// TIA Portal V17 export
// export: Created 2025-03-07T09:16:39.2442536Z, ExportSetting WithDefaults, DisplayName Totally Integrated Automation Portal, DisplayVersion V17 Update 8, DisplayName TIA Portal Openness, DisplayVersion V17 Update 8, DisplayName TIA Portal Version Control Interface, DisplayVersion V17, DisplayName SINAMICS Startdrive Advanced, DisplayVersion V17 SP2, DisplayName SINAMICS Startdrive G110M, G120, G120C, G120D, G120P, G115D, DisplayVersion V17 SP2, DisplayName SINAMICS Startdrive G130, G150, S120, S150, SINAMICS MV, S210, DisplayVersion V17 SP2, DisplayName STEP 7 Professional, DisplayVersion V17 Update 8, DisplayName SINUMERIK ONE STEP 7 Toolbox, DisplayVersion V17 Update 12, DisplayName SINUMERIK 840D sl STEP 7 Toolbox, DisplayVersion V17 Update 12, DisplayName STEP 7 Safety, DisplayVersion V17 Update 6, DisplayName WinCC Advanced, DisplayVersion V17 Update 8
DATA_BLOCK "DB2410_PLC_CNC_SIGNALS"   // DB2410
{ S7_Optimized_Access := 'FALSE'; DB_Accessible_From_OPC_UA := 'FALSE' }
AUTHOR : ETXETAR
VERSION : 1.0
// stored: AutoNumber false, DBAccessibleFromOPCUA false, DBAccessibleFromWebserver true, IsOnlyStoredInLoadMemory false, IsWriteProtectedInAS false
   VAR RETAIN
      PLC_NC_SIGNALS_1_32 : Struct   // NCK INPUTS EXTENSION BIT 41-72 / PLC NC SIGNALS BIT 1-32
         PLC_NC_SIGNAL_1 : Bool;   // NCK INPUTS EXTENSION 41 / PLC NC SIGNAL 1
         PLC_NC_SIGNAL_2 : Bool;   // NCK INPUTS EXTENSION 42 / PLC NC SIGNAL 2
         PLC_NC_SIGNAL_3 : Bool;   // NCK INPUTS EXTENSION 43 / PLC NC SIGNAL 3
         PLC_NC_SIGNAL_4 : Bool;   // NCK INPUTS EXTENSION 44 / PLC NC SIGNAL 4
         PLC_NC_SIGNAL_5 : Bool;   // NCK INPUTS EXTENSION 45 / PLC NC SIGNAL 5
         PLC_NC_SIGNAL_6 : Bool;   // NCK INPUTS EXTENSION 46 / PLC NC SIGNAL 6
         PLC_NC_SIGNAL_7 : Bool;   // NCK INPUTS EXTENSION 47 / PLC NC SIGNAL 7
         PLC_NC_SIGNAL_8 : Bool;   // NCK INPUTS EXTENSION 48 / PLC NC SIGNAL 8
         PLC_NC_SIGNAL_9 : Bool;   // NCK INPUTS EXTENSION 49 / PLC NC SIGNAL 9
         PLC_NC_SIGNAL_10 : Bool;   // NCK INPUTS EXTENSION 50 / PLC NC SIGNAL 10
         PLC_NC_SIGNAL_11 : Bool;   // NCK INPUTS EXTENSION 51 / PLC NC SIGNAL 11
         PLC_NC_SIGNAL_12 : Bool;   // NCK INPUTS EXTENSION 52 / PLC NC SIGNAL 12
         PLC_NC_SIGNAL_13 : Bool;   // NCK INPUTS EXTENSION 53 / PLC NC SIGNAL 13
         PLC_NC_SIGNAL_14 : Bool;   // NCK INPUTS EXTENSION 54 / PLC NC SIGNAL 14
         PLC_NC_SIGNAL_15 : Bool;   // NCK INPUTS EXTENSION 55 / PLC NC SIGNAL 15
         PLC_NC_SIGNAL_16 : Bool;   // NCK INPUTS EXTENSION 56 / PLC NC SIGNAL 16
         PLC_NC_SIGNAL_17 : Bool;   // NCK INPUTS EXTENSION 57 / PLC NC SIGNAL 17
         PLC_NC_SIGNAL_18 : Bool;   // NCK INPUTS EXTENSION 58 / PLC NC SIGNAL 18
         PLC_NC_SIGNAL_19 : Bool;   // NCK INPUTS EXTENSION 59 / PLC NC SIGNAL 19
         PLC_NC_SIGNAL_20 : Bool;   // NCK INPUTS EXTENSION 60 / PLC NC SIGNAL 20
         PLC_NC_SIGNAL_21 : Bool;   // NCK INPUTS EXTENSION 61 / PLC NC SIGNAL 21
         PLC_NC_SIGNAL_22 : Bool;   // NCK INPUTS EXTENSION 62 / PLC NC SIGNAL 22
         PLC_NC_SIGNAL_23 : Bool;   // NCK INPUTS EXTENSION 63 / PLC NC SIGNAL 23
         PLC_NC_SIGNAL_24 : Bool;   // NCK INPUTS EXTENSION 64 / PLC NC SIGNAL 24
         PLC_NC_SIGNAL_25 : Bool;   // NCK INPUTS EXTENSION 65 / PLC NC SIGNAL 25
         PLC_NC_SIGNAL_26 : Bool;   // NCK INPUTS EXTENSION 66 / PLC NC SIGNAL 26
         PLC_NC_SIGNAL_27 : Bool;   // NCK INPUTS EXTENSION 67 / PLC NC SIGNAL 27
         PLC_NC_SIGNAL_28 : Bool;   // NCK INPUTS EXTENSION 68 / PLC NC SIGNAL 28
         PLC_NC_SIGNAL_29 : Bool;   // NCK INPUTS EXTENSION 69 / PLC NC SIGNAL 29
         PLC_NC_SIGNAL_30 : Bool;   // NCK INPUTS EXTENSION 70 / PLC NC SIGNAL 30
         PLC_NC_SIGNAL_31 : Bool;   // NCK INPUTS EXTENSION 71 / PLC NC SIGNAL 31
         PLC_NC_SIGNAL_32 : Bool;   // NCK INPUTS EXTENSION 72 / PLC NC SIGNAL 32
      END_STRUCT;
      PLC_NC_SIGNALS_33_64 : Struct   // NCK INPUTS EXTENSION BIT 73-104 / PLC NC SIGNALS BIT 33-64
         PLC_NC_SIGNAL_33 : Bool;   // NCK INPUTS EXTENSION 73 / PLC NC SIGNAL 33
         PLC_NC_SIGNAL_34 : Bool;   // NCK INPUTS EXTENSION 74 / PLC NC SIGNAL 34
         PLC_NC_SIGNAL_35 : Bool;   // NCK INPUTS EXTENSION 75 / PLC NC SIGNAL 35
         PLC_NC_SIGNAL_36 : Bool;   // NCK INPUTS EXTENSION 76 / PLC NC SIGNAL 36
         PLC_NC_SIGNAL_37 : Bool;   // NCK INPUTS EXTENSION 77 / PLC NC SIGNAL 37
         PLC_NC_SIGNAL_38 : Bool;   // NCK INPUTS EXTENSION 78 / PLC NC SIGNAL 38
         PLC_NC_SIGNAL_39 : Bool;   // NCK INPUTS EXTENSION 79 / PLC NC SIGNAL 39
         PLC_NC_SIGNAL_40 : Bool;   // NCK INPUTS EXTENSION 80 / PLC NC SIGNAL 40
         PLC_NC_SIGNAL_41 : Bool;   // NCK INPUTS EXTENSION 81 / PLC NC SIGNAL 41
         PLC_NC_SIGNAL_42 : Bool;   // NCK INPUTS EXTENSION 82 / PLC NC SIGNAL 42
         PLC_NC_SIGNAL_43 : Bool;   // NCK INPUTS EXTENSION 83 / PLC NC SIGNAL 43
         PLC_NC_SIGNAL_44 : Bool;   // NCK INPUTS EXTENSION 84 / PLC NC SIGNAL 44
         PLC_NC_SIGNAL_45 : Bool;   // NCK INPUTS EXTENSION 85 / PLC NC SIGNAL 45
         PLC_NC_SIGNAL_46 : Bool;   // NCK INPUTS EXTENSION 86 / PLC NC SIGNAL 46
         PLC_NC_SIGNAL_47 : Bool;   // NCK INPUTS EXTENSION 87 / PLC NC SIGNAL 47
         PLC_NC_SIGNAL_48 : Bool;   // NCK INPUTS EXTENSION 88 / PLC NC SIGNAL 48
         PLC_NC_SIGNAL_49 : Bool;   // NCK INPUTS EXTENSION 89 / PLC NC SIGNAL 49
         PLC_NC_SIGNAL_50 : Bool;   // NCK INPUTS EXTENSION 90 / PLC NC SIGNAL 50
         PLC_NC_SIGNAL_51 : Bool;   // NCK INPUTS EXTENSION 91 / PLC NC SIGNAL 51
         PLC_NC_SIGNAL_52 : Bool;   // NCK INPUTS EXTENSION 92 / PLC NC SIGNAL 52
         PLC_NC_SIGNAL_53 : Bool;   // NCK INPUTS EXTENSION 93 / PLC NC SIGNAL 53
         PLC_NC_SIGNAL_54 : Bool;   // NCK INPUTS EXTENSION 94 / PLC NC SIGNAL 54
         PLC_NC_SIGNAL_55 : Bool;   // NCK INPUTS EXTENSION 95 / PLC NC SIGNAL 55
         PLC_NC_SIGNAL_56 : Bool;   // NCK INPUTS EXTENSION 96 / PLC NC SIGNAL 56
         PLC_NC_SIGNAL_57 : Bool;   // NCK INPUTS EXTENSION 97 / PLC NC SIGNAL 57
         PLC_NC_SIGNAL_58 : Bool;   // NCK INPUTS EXTENSION 98 / PLC NC SIGNAL 58
         PLC_NC_SIGNAL_59 : Bool;   // NCK INPUTS EXTENSION 99 / PLC NC SIGNAL 59
         PLC_NC_SIGNAL_60 : Bool;   // NCK INPUTS EXTENSION 100 / PLC NC SIGNAL 60
         PLC_NC_SIGNAL_61 : Bool;   // NCK INPUTS EXTENSION 101 / PLC NC SIGNAL 61
         PLC_NC_SIGNAL_62 : Bool;   // NCK INPUTS EXTENSION 102 / PLC NC SIGNAL 62
         PLC_NC_SIGNAL_63 : Bool;   // NCK INPUTS EXTENSION 103 / PLC NC SIGNAL 63
         PLC_NC_SIGNAL_64 : Bool;   // NCK INPUTS EXTENSION 104 / PLC NC SIGNAL 64
      END_STRUCT;
      PLC_NC_SIGNALS_65_96 : Struct   // NCK INPUTS EXTENSION BIT 73-104 / PLC NC SIGNALS BIT 65-96
         PLC_NC_SIGNAL_65 : Bool;   // NCK INPUTS EXTENSION 73 / PLC NC SIGNAL 65
         PLC_NC_SIGNAL_66 : Bool;   // NCK INPUTS EXTENSION 74 / PLC NC SIGNAL 66
         PLC_NC_SIGNAL_67 : Bool;   // NCK INPUTS EXTENSION 75 / PLC NC SIGNAL 67
         PLC_NC_SIGNAL_68 : Bool;   // NCK INPUTS EXTENSION 76 / PLC NC SIGNAL 68
         PLC_NC_SIGNAL_69 : Bool;   // NCK INPUTS EXTENSION 77 / PLC NC SIGNAL 69
         PLC_NC_SIGNAL_70 : Bool;   // NCK INPUTS EXTENSION 78 / PLC NC SIGNAL 70
         PLC_NC_SIGNAL_71 : Bool;   // NCK INPUTS EXTENSION 79 / PLC NC SIGNAL 71
         PLC_NC_SIGNAL_72 : Bool;   // NCK INPUTS EXTENSION 80 / PLC NC SIGNAL 72
         PLC_NC_SIGNAL_73 : Bool;   // NCK INPUTS EXTENSION 81 / PLC NC SIGNAL 73
         PLC_NC_SIGNAL_74 : Bool;   // NCK INPUTS EXTENSION 82 / PLC NC SIGNAL 74
         PLC_NC_SIGNAL_75 : Bool;   // NCK INPUTS EXTENSION 83 / PLC NC SIGNAL 75
         PLC_NC_SIGNAL_76 : Bool;   // NCK INPUTS EXTENSION 84 / PLC NC SIGNAL 76
         PLC_NC_SIGNAL_77 : Bool;   // NCK INPUTS EXTENSION 85 / PLC NC SIGNAL 77
         PLC_NC_SIGNAL_78 : Bool;   // NCK INPUTS EXTENSION 86 / PLC NC SIGNAL 78
         PLC_NC_SIGNAL_79 : Bool;   // NCK INPUTS EXTENSION 87 / PLC NC SIGNAL 79
         PLC_NC_SIGNAL_80 : Bool;   // NCK INPUTS EXTENSION 88 / PLC NC SIGNAL 80
         PLC_NC_SIGNAL_81 : Bool;   // NCK INPUTS EXTENSION 89 / PLC NC SIGNAL 81
         PLC_NC_SIGNAL_82 : Bool;   // NCK INPUTS EXTENSION 90 / PLC NC SIGNAL 82
         PLC_NC_SIGNAL_83 : Bool;   // NCK INPUTS EXTENSION 91 / PLC NC SIGNAL 83
         PLC_NC_SIGNAL_84 : Bool;   // NCK INPUTS EXTENSION 92 / PLC NC SIGNAL 84
         PLC_NC_SIGNAL_85 : Bool;   // NCK INPUTS EXTENSION 93 / PLC NC SIGNAL 85
         PLC_NC_SIGNAL_86 : Bool;   // NCK INPUTS EXTENSION 94 / PLC NC SIGNAL 86
         PLC_NC_SIGNAL_87 : Bool;   // NCK INPUTS EXTENSION 95 / PLC NC SIGNAL 87
         PLC_NC_SIGNAL_88 : Bool;   // NCK INPUTS EXTENSION 96 / PLC NC SIGNAL 88
         PLC_NC_SIGNAL_89 : Bool;   // NCK INPUTS EXTENSION 97 / PLC NC SIGNAL 89
         PLC_NC_SIGNAL_90 : Bool;   // NCK INPUTS EXTENSION 98 / PLC NC SIGNAL 90
         PLC_NC_SIGNAL_91 : Bool;   // NCK INPUTS EXTENSION 99 / PLC NC SIGNAL 91
         PLC_NC_SIGNAL_92 : Bool;   // NCK INPUTS EXTENSION 100 / PLC NC SIGNAL 92
         PLC_NC_SIGNAL_93 : Bool;   // NCK INPUTS EXTENSION 101 / PLC NC SIGNAL 93
         PLC_NC_SIGNAL_94 : Bool;   // NCK INPUTS EXTENSION 102 / PLC NC SIGNAL 94
         PLC_NC_SIGNAL_95 : Bool;   // NCK INPUTS EXTENSION 103 / PLC NC SIGNAL 95
         PLC_NC_SIGNAL_96 : Bool;   // NCK INPUTS EXTENSION 104 / PLC NC SIGNAL 96
      END_STRUCT;
      PLC_NC_SIGNALS_97_128 : Struct   // NCK INPUTS EXTENSION BIT 73-104 / PLC NC SIGNALS BIT 97-128
         PLC_NC_SIGNAL_97 : Bool;   // NCK INPUTS EXTENSION 73 / PLC NC SIGNAL 97
         PLC_NC_SIGNAL_98 : Bool;   // NCK INPUTS EXTENSION 74 / PLC NC SIGNAL 98
         PLC_NC_SIGNAL_99 : Bool;   // NCK INPUTS EXTENSION 75 / PLC NC SIGNAL 99
         PLC_NC_SIGNAL_100 : Bool;   // NCK INPUTS EXTENSION 76 / PLC NC SIGNAL 100
         PLC_NC_SIGNAL_101 : Bool;   // NCK INPUTS EXTENSION 77 / PLC NC SIGNAL 101
         PLC_NC_SIGNAL_102 : Bool;   // NCK INPUTS EXTENSION 78 / PLC NC SIGNAL 102
         PLC_NC_SIGNAL_103 : Bool;   // NCK INPUTS EXTENSION 79 / PLC NC SIGNAL 103
         PLC_NC_SIGNAL_104 : Bool;   // NCK INPUTS EXTENSION 80 / PLC NC SIGNAL 104
         PLC_NC_SIGNAL_105 : Bool;   // NCK INPUTS EXTENSION 81 / PLC NC SIGNAL 105
         PLC_NC_SIGNAL_106 : Bool;   // NCK INPUTS EXTENSION 82 / PLC NC SIGNAL 106
         PLC_NC_SIGNAL_107 : Bool;   // NCK INPUTS EXTENSION 83 / PLC NC SIGNAL 107
         PLC_NC_SIGNAL_108 : Bool;   // NCK INPUTS EXTENSION 84 / PLC NC SIGNAL 108
         PLC_NC_SIGNAL_109 : Bool;   // NCK INPUTS EXTENSION 85 / PLC NC SIGNAL 109
         PLC_NC_SIGNAL_110 : Bool;   // NCK INPUTS EXTENSION 86 / PLC NC SIGNAL 110
         PLC_NC_SIGNAL_111 : Bool;   // NCK INPUTS EXTENSION 87 / PLC NC SIGNAL 111
         PLC_NC_SIGNAL_112 : Bool;   // NCK INPUTS EXTENSION 88 / PLC NC SIGNAL 112
         PLC_NC_SIGNAL_113 : Bool;   // NCK INPUTS EXTENSION 89 / PLC NC SIGNAL 113
         PLC_NC_SIGNAL_114 : Bool;   // NCK INPUTS EXTENSION 90 / PLC NC SIGNAL 114
         PLC_NC_SIGNAL_115 : Bool;   // NCK INPUTS EXTENSION 91 / PLC NC SIGNAL 115
         PLC_NC_SIGNAL_116 : Bool;   // NCK INPUTS EXTENSION 92 / PLC NC SIGNAL 116
         PLC_NC_SIGNAL_117 : Bool;   // NCK INPUTS EXTENSION 93 / PLC NC SIGNAL 117
         PLC_NC_SIGNAL_118 : Bool;   // NCK INPUTS EXTENSION 94 / PLC NC SIGNAL 118
         PLC_NC_SIGNAL_119 : Bool;   // NCK INPUTS EXTENSION 95 / PLC NC SIGNAL 119
         PLC_NC_SIGNAL_120 : Bool;   // NCK INPUTS EXTENSION 96 / PLC NC SIGNAL 120
         PLC_NC_SIGNAL_121 : Bool;   // NCK INPUTS EXTENSION 97 / PLC NC SIGNAL 121
         PLC_NC_SIGNAL_122 : Bool;   // NCK INPUTS EXTENSION 98 / PLC NC SIGNAL 122
         PLC_NC_SIGNAL_123 : Bool;   // NCK INPUTS EXTENSION 99 / PLC NC SIGNAL 123
         PLC_NC_SIGNAL_124 : Bool;   // NCK INPUTS EXTENSION 100 / PLC NC SIGNAL 124
         PLC_NC_SIGNAL_125 : Bool;   // NCK INPUTS EXTENSION 101 / PLC NC SIGNAL 125
         PLC_NC_SIGNAL_126 : Bool;   // NCK INPUTS EXTENSION 102 / PLC NC SIGNAL 126
         PLC_NC_SIGNAL_127 : Bool;   // NCK INPUTS EXTENSION 103 / PLC NC SIGNAL 127
         PLC_NC_SIGNAL_128 : Bool;   // NCK INPUTS EXTENSION 104 / PLC NC SIGNAL 128
      END_STRUCT;
      PLC_NC_SIGNALS_129_160 : Struct   // NCK INPUTS EXTENSION BIT 73-104 / PLC NC SIGNALS BIT 129-160
         PLC_NC_SIGNAL_129 : Bool;   // NCK INPUTS EXTENSION 73 / PLC NC SIGNAL 129
         PLC_NC_SIGNAL_130 : Bool;   // NCK INPUTS EXTENSION 74 / PLC NC SIGNAL 130
         PLC_NC_SIGNAL_131 : Bool;   // NCK INPUTS EXTENSION 75 / PLC NC SIGNAL 131
         PLC_NC_SIGNAL_132 : Bool;   // NCK INPUTS EXTENSION 76 / PLC NC SIGNAL 132
         PLC_NC_SIGNAL_133 : Bool;   // NCK INPUTS EXTENSION 77 / PLC NC SIGNAL 133
         PLC_NC_SIGNAL_134 : Bool;   // NCK INPUTS EXTENSION 78 / PLC NC SIGNAL 134
         PLC_NC_SIGNAL_135 : Bool;   // NCK INPUTS EXTENSION 79 / PLC NC SIGNAL 135
         PLC_NC_SIGNAL_136 : Bool;   // NCK INPUTS EXTENSION 80 / PLC NC SIGNAL 136
         PLC_NC_SIGNAL_137 : Bool;   // NCK INPUTS EXTENSION 81 / PLC NC SIGNAL 137
         PLC_NC_SIGNAL_138 : Bool;   // NCK INPUTS EXTENSION 82 / PLC NC SIGNAL 138
         PLC_NC_SIGNAL_139 : Bool;   // NCK INPUTS EXTENSION 83 / PLC NC SIGNAL 139
         PLC_NC_SIGNAL_140 : Bool;   // NCK INPUTS EXTENSION 84 / PLC NC SIGNAL 140
         PLC_NC_SIGNAL_141 : Bool;   // NCK INPUTS EXTENSION 85 / PLC NC SIGNAL 141
         PLC_NC_SIGNAL_142 : Bool;   // NCK INPUTS EXTENSION 86 / PLC NC SIGNAL 142
         PLC_NC_SIGNAL_143 : Bool;   // NCK INPUTS EXTENSION 87 / PLC NC SIGNAL 143
         PLC_NC_SIGNAL_144 : Bool;   // NCK INPUTS EXTENSION 88 / PLC NC SIGNAL 144
         PLC_NC_SIGNAL_145 : Bool;   // NCK INPUTS EXTENSION 89 / PLC NC SIGNAL 145
         PLC_NC_SIGNAL_146 : Bool;   // NCK INPUTS EXTENSION 90 / PLC NC SIGNAL 146
         PLC_NC_SIGNAL_147 : Bool;   // NCK INPUTS EXTENSION 91 / PLC NC SIGNAL 147
         PLC_NC_SIGNAL_148 : Bool;   // NCK INPUTS EXTENSION 92 / PLC NC SIGNAL 148
         PLC_NC_SIGNAL_149 : Bool;   // NCK INPUTS EXTENSION 93 / PLC NC SIGNAL 149
         PLC_NC_SIGNAL_150 : Bool;   // NCK INPUTS EXTENSION 94 / PLC NC SIGNAL 150
         PLC_NC_SIGNAL_151 : Bool;   // NCK INPUTS EXTENSION 95 / PLC NC SIGNAL 151
         PLC_NC_SIGNAL_152 : Bool;   // NCK INPUTS EXTENSION 96 / PLC NC SIGNAL 152
         PLC_NC_SIGNAL_153 : Bool;   // NCK INPUTS EXTENSION 97 / PLC NC SIGNAL 153
         PLC_NC_SIGNAL_154 : Bool;   // NCK INPUTS EXTENSION 98 / PLC NC SIGNAL 154
         PLC_NC_SIGNAL_155 : Bool;   // NCK INPUTS EXTENSION 99 / PLC NC SIGNAL 155
         PLC_NC_SIGNAL_156 : Bool;   // NCK INPUTS EXTENSION 100 / PLC NC SIGNAL 156
         PLC_NC_SIGNAL_157 : Bool;   // NCK INPUTS EXTENSION 101 / PLC NC SIGNAL 157
         PLC_NC_SIGNAL_158 : Bool;   // NCK INPUTS EXTENSION 102 / PLC NC SIGNAL 158
         PLC_NC_SIGNAL_159 : Bool;   // NCK INPUTS EXTENSION 103 / PLC NC SIGNAL 159
         PLC_NC_SIGNAL_160 : Bool;   // NCK INPUTS EXTENSION 104 / PLC NC SIGNAL 160
      END_STRUCT;
      PLC_NC_SIGNALS_161_192 : Struct   // NCK INPUTS EXTENSION BIT 73-104 / PLC NC SIGNALS BIT 161-192
         PLC_NC_SIGNAL_161 : Bool;   // NCK INPUTS EXTENSION 73 / PLC NC SIGNAL 161
         PLC_NC_SIGNAL_162 : Bool;   // NCK INPUTS EXTENSION 74 / PLC NC SIGNAL 162
         PLC_NC_SIGNAL_163 : Bool;   // NCK INPUTS EXTENSION 75 / PLC NC SIGNAL 163
         PLC_NC_SIGNAL_164 : Bool;   // NCK INPUTS EXTENSION 76 / PLC NC SIGNAL 164
         PLC_NC_SIGNAL_165 : Bool;   // NCK INPUTS EXTENSION 77 / PLC NC SIGNAL 165
         PLC_NC_SIGNAL_166 : Bool;   // NCK INPUTS EXTENSION 78 / PLC NC SIGNAL 166
         PLC_NC_SIGNAL_167 : Bool;   // NCK INPUTS EXTENSION 79 / PLC NC SIGNAL 167
         PLC_NC_SIGNAL_168 : Bool;   // NCK INPUTS EXTENSION 80 / PLC NC SIGNAL 168
         PLC_NC_SIGNAL_169 : Bool;   // NCK INPUTS EXTENSION 81 / PLC NC SIGNAL 169
         PLC_NC_SIGNAL_170 : Bool;   // NCK INPUTS EXTENSION 82 / PLC NC SIGNAL 170
         PLC_NC_SIGNAL_171 : Bool;   // NCK INPUTS EXTENSION 83 / PLC NC SIGNAL 171
         PLC_NC_SIGNAL_172 : Bool;   // NCK INPUTS EXTENSION 84 / PLC NC SIGNAL 172
         PLC_NC_SIGNAL_173 : Bool;   // NCK INPUTS EXTENSION 85 / PLC NC SIGNAL 173
         PLC_NC_SIGNAL_174 : Bool;   // NCK INPUTS EXTENSION 86 / PLC NC SIGNAL 174
         PLC_NC_SIGNAL_175 : Bool;   // NCK INPUTS EXTENSION 87 / PLC NC SIGNAL 175
         PLC_NC_SIGNAL_176 : Bool;   // NCK INPUTS EXTENSION 88 / PLC NC SIGNAL 176
         PLC_NC_SIGNAL_177 : Bool;   // NCK INPUTS EXTENSION 89 / PLC NC SIGNAL 177
         PLC_NC_SIGNAL_178 : Bool;   // NCK INPUTS EXTENSION 90 / PLC NC SIGNAL 178
         PLC_NC_SIGNAL_179 : Bool;   // NCK INPUTS EXTENSION 91 / PLC NC SIGNAL 179
         PLC_NC_SIGNAL_180 : Bool;   // NCK INPUTS EXTENSION 92 / PLC NC SIGNAL 180
         PLC_NC_SIGNAL_181 : Bool;   // NCK INPUTS EXTENSION 93 / PLC NC SIGNAL 181
         PLC_NC_SIGNAL_182 : Bool;   // NCK INPUTS EXTENSION 94 / PLC NC SIGNAL 182
         PLC_NC_SIGNAL_183 : Bool;   // NCK INPUTS EXTENSION 95 / PLC NC SIGNAL 183
         PLC_NC_SIGNAL_184 : Bool;   // NCK INPUTS EXTENSION 96 / PLC NC SIGNAL 184
         PLC_NC_SIGNAL_185 : Bool;   // NCK INPUTS EXTENSION 97 / PLC NC SIGNAL 185
         PLC_NC_SIGNAL_186 : Bool;   // NCK INPUTS EXTENSION 98 / PLC NC SIGNAL 186
         PLC_NC_SIGNAL_187 : Bool;   // NCK INPUTS EXTENSION 99 / PLC NC SIGNAL 187
         PLC_NC_SIGNAL_188 : Bool;   // NCK INPUTS EXTENSION 100 / PLC NC SIGNAL 188
         PLC_NC_SIGNAL_189 : Bool;   // NCK INPUTS EXTENSION 101 / PLC NC SIGNAL 189
         PLC_NC_SIGNAL_190 : Bool;   // NCK INPUTS EXTENSION 102 / PLC NC SIGNAL 190
         PLC_NC_SIGNAL_191 : Bool;   // NCK INPUTS EXTENSION 103 / PLC NC SIGNAL 191
         PLC_NC_SIGNAL_192 : Bool;   // NCK INPUTS EXTENSION 104 / PLC NC SIGNAL 192
      END_STRUCT;
      PLC_NC_SIGNALS_193_224 : Struct   // NCK INPUTS EXTENSION BIT 73-104 / PLC NC SIGNALS BIT 193-224
         PLC_NC_SIGNAL_193 : Bool;   // NCK INPUTS EXTENSION 73 / PLC NC SIGNAL 193
         PLC_NC_SIGNAL_194 : Bool;   // NCK INPUTS EXTENSION 74 / PLC NC SIGNAL 194
         PLC_NC_SIGNAL_195 : Bool;   // NCK INPUTS EXTENSION 75 / PLC NC SIGNAL 195
         PLC_NC_SIGNAL_196 : Bool;   // NCK INPUTS EXTENSION 76 / PLC NC SIGNAL 196
         PLC_NC_SIGNAL_197 : Bool;   // NCK INPUTS EXTENSION 77 / PLC NC SIGNAL 197
         PLC_NC_SIGNAL_198 : Bool;   // NCK INPUTS EXTENSION 78 / PLC NC SIGNAL 198
         PLC_NC_SIGNAL_199 : Bool;   // NCK INPUTS EXTENSION 79 / PLC NC SIGNAL 199
         PLC_NC_SIGNAL_200 : Bool;   // NCK INPUTS EXTENSION 80 / PLC NC SIGNAL 200
         PLC_NC_SIGNAL_201 : Bool;   // NCK INPUTS EXTENSION 81 / PLC NC SIGNAL 201
         PLC_NC_SIGNAL_202 : Bool;   // NCK INPUTS EXTENSION 82 / PLC NC SIGNAL 202
         PLC_NC_SIGNAL_203 : Bool;   // NCK INPUTS EXTENSION 83 / PLC NC SIGNAL 203
         PLC_NC_SIGNAL_204 : Bool;   // NCK INPUTS EXTENSION 84 / PLC NC SIGNAL 204
         PLC_NC_SIGNAL_205 : Bool;   // NCK INPUTS EXTENSION 85 / PLC NC SIGNAL 205
         PLC_NC_SIGNAL_206 : Bool;   // NCK INPUTS EXTENSION 86 / PLC NC SIGNAL 206
         PLC_NC_SIGNAL_207 : Bool;   // NCK INPUTS EXTENSION 87 / PLC NC SIGNAL 207
         PLC_NC_SIGNAL_208 : Bool;   // NCK INPUTS EXTENSION 88 / PLC NC SIGNAL 208
         PLC_NC_SIGNAL_209 : Bool;   // NCK INPUTS EXTENSION 89 / PLC NC SIGNAL 209
         PLC_NC_SIGNAL_210 : Bool;   // NCK INPUTS EXTENSION 90 / PLC NC SIGNAL 210
         PLC_NC_SIGNAL_211 : Bool;   // NCK INPUTS EXTENSION 91 / PLC NC SIGNAL 211
         PLC_NC_SIGNAL_212 : Bool;   // NCK INPUTS EXTENSION 92 / PLC NC SIGNAL 212
         PLC_NC_SIGNAL_213 : Bool;   // NCK INPUTS EXTENSION 93 / PLC NC SIGNAL 213
         PLC_NC_SIGNAL_214 : Bool;   // NCK INPUTS EXTENSION 94 / PLC NC SIGNAL 214
         PLC_NC_SIGNAL_215 : Bool;   // NCK INPUTS EXTENSION 95 / PLC NC SIGNAL 215
         PLC_NC_SIGNAL_216 : Bool;   // NCK INPUTS EXTENSION 96 / PLC NC SIGNAL 216
         PLC_NC_SIGNAL_217 : Bool;   // NCK INPUTS EXTENSION 97 / PLC NC SIGNAL 217
         PLC_NC_SIGNAL_218 : Bool;   // NCK INPUTS EXTENSION 98 / PLC NC SIGNAL 218
         PLC_NC_SIGNAL_219 : Bool;   // NCK INPUTS EXTENSION 99 / PLC NC SIGNAL 219
         PLC_NC_SIGNAL_220 : Bool;   // NCK INPUTS EXTENSION 100 / PLC NC SIGNAL 220
         PLC_NC_SIGNAL_221 : Bool;   // NCK INPUTS EXTENSION 101 / PLC NC SIGNAL 221
         PLC_NC_SIGNAL_222 : Bool;   // NCK INPUTS EXTENSION 102 / PLC NC SIGNAL 222
         PLC_NC_SIGNAL_223 : Bool;   // NCK INPUTS EXTENSION 103 / PLC NC SIGNAL 223
         PLC_NC_SIGNAL_224 : Bool;   // NCK INPUTS EXTENSION 104 / PLC NC SIGNAL 224
      END_STRUCT;
      PLC_NC_SIGNALS_225_256 : Struct   // NCK INPUTS EXTENSION BIT 73-104 / PLC NC SIGNALS BIT 225-256
         PLC_NC_SIGNAL_225 : Bool;   // NCK INPUTS EXTENSION 73 / PLC NC SIGNAL 225
         PLC_NC_SIGNAL_226 : Bool;   // NCK INPUTS EXTENSION 74 / PLC NC SIGNAL 226
         PLC_NC_SIGNAL_227 : Bool;   // NCK INPUTS EXTENSION 75 / PLC NC SIGNAL 227
         PLC_NC_SIGNAL_228 : Bool;   // NCK INPUTS EXTENSION 76 / PLC NC SIGNAL 228
         PLC_NC_SIGNAL_229 : Bool;   // NCK INPUTS EXTENSION 77 / PLC NC SIGNAL 229
         PLC_NC_SIGNAL_230 : Bool;   // NCK INPUTS EXTENSION 78 / PLC NC SIGNAL 230
         PLC_NC_SIGNAL_231 : Bool;   // NCK INPUTS EXTENSION 79 / PLC NC SIGNAL 231
         PLC_NC_SIGNAL_232 : Bool;   // NCK INPUTS EXTENSION 80 / PLC NC SIGNAL 232
         PLC_NC_SIGNAL_233 : Bool;   // NCK INPUTS EXTENSION 81 / PLC NC SIGNAL 233
         PLC_NC_SIGNAL_234 : Bool;   // NCK INPUTS EXTENSION 82 / PLC NC SIGNAL 234
         PLC_NC_SIGNAL_235 : Bool;   // NCK INPUTS EXTENSION 83 / PLC NC SIGNAL 235
         PLC_NC_SIGNAL_236 : Bool;   // NCK INPUTS EXTENSION 84 / PLC NC SIGNAL 236
         PLC_NC_SIGNAL_237 : Bool;   // NCK INPUTS EXTENSION 85 / PLC NC SIGNAL 237
         PLC_NC_SIGNAL_238 : Bool;   // NCK INPUTS EXTENSION 86 / PLC NC SIGNAL 238
         PLC_NC_SIGNAL_239 : Bool;   // NCK INPUTS EXTENSION 87 / PLC NC SIGNAL 239
         PLC_NC_SIGNAL_240 : Bool;   // NCK INPUTS EXTENSION 88 / PLC NC SIGNAL 240
         PLC_NC_SIGNAL_241 : Bool;   // NCK INPUTS EXTENSION 89 / PLC NC SIGNAL 241
         PLC_NC_SIGNAL_242 : Bool;   // NCK INPUTS EXTENSION 90 / PLC NC SIGNAL 242
         PLC_NC_SIGNAL_243 : Bool;   // NCK INPUTS EXTENSION 91 / PLC NC SIGNAL 243
         PLC_NC_SIGNAL_244 : Bool;   // NCK INPUTS EXTENSION 92 / PLC NC SIGNAL 244
         PLC_NC_SIGNAL_245 : Bool;   // NCK INPUTS EXTENSION 93 / PLC NC SIGNAL 245
         PLC_NC_SIGNAL_246 : Bool;   // NCK INPUTS EXTENSION 94 / PLC NC SIGNAL 246
         PLC_NC_SIGNAL_247 : Bool;   // NCK INPUTS EXTENSION 95 / PLC NC SIGNAL 247
         PLC_NC_SIGNAL_248 : Bool;   // NCK INPUTS EXTENSION 96 / PLC NC SIGNAL 248
         PLC_NC_SIGNAL_249 : Bool;   // NCK INPUTS EXTENSION 97 / PLC NC SIGNAL 249
         PLC_NC_SIGNAL_250 : Bool;   // NCK INPUTS EXTENSION 98 / PLC NC SIGNAL 250
         PLC_NC_SIGNAL_251 : Bool;   // NCK INPUTS EXTENSION 99 / PLC NC SIGNAL 251
         PLC_NC_SIGNAL_252 : Bool;   // NCK INPUTS EXTENSION 100 / PLC NC SIGNAL 252
         PLC_NC_SIGNAL_253 : Bool;   // NCK INPUTS EXTENSION 101 / PLC NC SIGNAL 253
         PLC_NC_SIGNAL_254 : Bool;   // NCK INPUTS EXTENSION 102 / PLC NC SIGNAL 254
         PLC_NC_SIGNAL_255 : Bool;   // NCK INPUTS EXTENSION 103 / PLC NC SIGNAL 255
         PLC_NC_SIGNAL_256 : Bool;   // NCK INPUTS EXTENSION 104 / PLC NC SIGNAL 256
      END_STRUCT;
      DBB_DBW_DBD_VAL_4000 : Int := 4000;   // NCK INPUTS EXTENSION BIT 41-72 / PLC NC SIGNALS BIT 1-32
      DBB_DBW_DBD_VAL_4001 : Int := 4001;
      DBB_DBW_DBD_VAL_4002 : Int := 4002;
      DBB_DBW_DBD_VAL_4003 : Int := 4003;
      DBB_DBW_DBD_VAL_4004 : Int := 4004;   // NCK INPUTS EXTENSION BIT 73-104 / PLC NC SIGNALS BIT 33-64
      DBB_DBW_DBD_VAL_4005 : Int := 4005;
      DBB_DBW_DBD_VAL_4006 : Int := 4006;
      DBB_DBW_DBD_VAL_4007 : Int := 4007;
      DBB_DBW_DBD_VAL_4008 : Int := 4008;   // PLC NC SIGNALS BIT 65-96
      DBB_DBW_DBD_VAL_4009 : Int := 4009;
      DBB_DBW_DBD_VAL_4010 : Int := 4010;
      DBB_DBW_DBD_VAL_4011 : Int := 4011;
      DBB_DBW_DBD_VAL_4012 : Int := 4012;   // PLC NC SIGNALS BIT 97-128
      DBB_DBW_DBD_VAL_4013 : Int := 4013;
      DBB_DBW_DBD_VAL_4014 : Int := 4014;
      DBB_DBW_DBD_VAL_4015 : Int := 4015;
      DBB_DBW_DBD_VAL_4016 : Int := 4016;   // PLC NC SIGNALS BIT 129-160
      DBB_DBW_DBD_VAL_4017 : Int := 4017;
      DBB_DBW_DBD_VAL_4018 : Int := 4018;
      DBB_DBW_DBD_VAL_4019 : Int := 4019;
      DBB_DBW_DBD_VAL_4020 : Int := 4020;   // PLC NC SIGNALS BIT 161-192
      DBB_DBW_DBD_VAL_4021 : Int := 4021;
      DBB_DBW_DBD_VAL_4022 : Int := 4022;
      DBB_DBW_DBD_VAL_4023 : Int := 4023;
      DBB_DBW_DBD_VAL_4024 : Int := 4024;   // PLC NC SIGNALS BIT 193-224
      DBB_DBW_DBD_VAL_4025 : Int := 4025;
      DBB_DBW_DBD_VAL_4026 : Int := 4026;
      DBB_DBW_DBD_VAL_4027 : Int := 4027;
      DBB_DBW_DBD_VAL_4028 : Int := 4028;   // PLC NC SIGNALS BIT 225-256
      DBB_DBW_DBD_VAL_4029 : Int := 4029;
      DBB_DBW_DBD_VAL_4030 : Int := 4030;
      DBB_DBW_DBD_VAL_4031 : Int := 4031;
   END_VAR
BEGIN
END_DATA_BLOCK
